SYSTEM DASDA12 (* System Configuration *)
  (* Standard: 61499-1 *)
  (* Version 0.4, 2009-03-05, JHC, Holobloc Inc., Deleted Application. *)
  (* Version 0.3, 2003-12-05, JHC, Rockwell Automation, Renamed from NEWSYSTEM. *)
  (* Version 0.2, 2002-11-05, JHC, Rockwell Automation, Fixed missing (empty) FBD in Application. *)
  (* Version 0.1, 2002-01-17, JHC, Rockwell Automation, Minor cleanup *)
  (* Version 0.0, 2000-05-27, JHC, Rockwell Automation *)
  DEVICE HMI_LAYER : FRAME_DEVICE(BOUNDS := [0,0,200,400])
    RESOURCE HMI : PANEL_RESOURCE(ROWS := 5, COLS := 1)
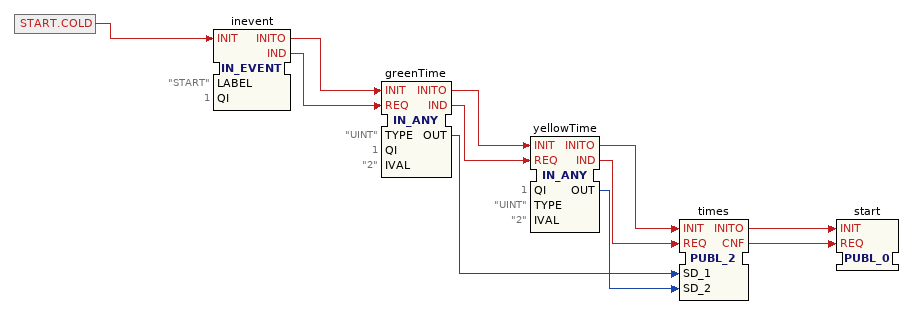
      FBS
        inevent : IN_EVENT(LABEL := "START", QI := 1);
        start : PUBL_0;
        greenTime : IN_ANY(TYPE := "UINT", QI := 1, IVAL := "2");
        yellowTime : IN_ANY(QI := 1, TYPE := "UINT", IVAL := "2");
        times : PUBL_2;
      END_FBS
      EVENT_CONNECTIONS
        START.COLD TO inevent.INIT;
        greenTime.INITO TO yellowTime.INIT;
        inevent.INITO TO greenTime.INIT;
        inevent.IND TO greenTime.REQ;
        yellowTime.INITO TO times.INIT;
        times.INITO TO start.INIT;
        times.CNF TO start.REQ;
        greenTime.IND TO yellowTime.REQ;
        yellowTime.IND TO times.REQ;
      END_CONNECTIONS
      DATA_CONNECTIONS
        greenTime.OUT TO times.SD_1;
        yellowTime.OUT TO times.SD_2;
      END_CONNECTIONS
    END_RESOURCE
  END_DEVICE
  DEVICE MODEL_LAYER : FRAME_DEVICE
    RESOURCE LIGHTS : PANEL_RESOURCE
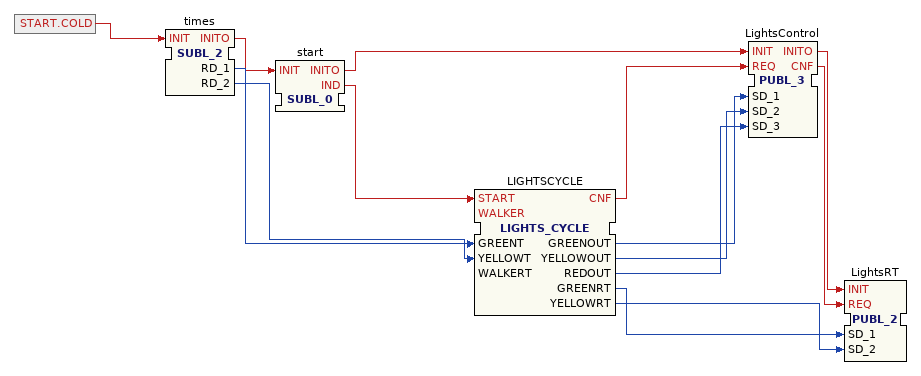
      FBS
        LightsControl : PUBL_3;
        start : SUBL_0;
        times : SUBL_2;
        LIGHTSCYCLE : LIGHTS_CYCLE;
        LightsRT : PUBL_2;
      END_FBS
      EVENT_CONNECTIONS
        START.COLD TO times.INIT;
        times.INITO TO start.INIT;
        start.INITO TO LightsControl.INIT;
        start.IND TO LIGHTSCYCLE.START;
        LIGHTSCYCLE.CNF TO LightsControl.REQ;
        LightsControl.INITO TO LightsRT.INIT;
        LightsControl.CNF TO LightsRT.REQ;
      END_CONNECTIONS
      DATA_CONNECTIONS
        LIGHTSCYCLE.GREENOUT TO LightsControl.SD_1;
        LIGHTSCYCLE.YELLOWOUT TO LightsControl.SD_2;
        LIGHTSCYCLE.REDOUT TO LightsControl.SD_3;
        LIGHTSCYCLE.GREENRT TO LightsRT.SD_1;
        LIGHTSCYCLE.YELLOWRT TO LightsRT.SD_2;
        times.RD_1 TO LIGHTSCYCLE.GREENT;
        times.RD_2 TO LIGHTSCYCLE.YELLOWT;
      END_CONNECTIONS
    END_RESOURCE
  END_DEVICE
  DEVICE VIEW_LAYER : FRAME_DEVICE(BOUNDS := [200,0,600,400], GRID := [1,1])
    RESOURCE view_res : PANEL_RESOURCE
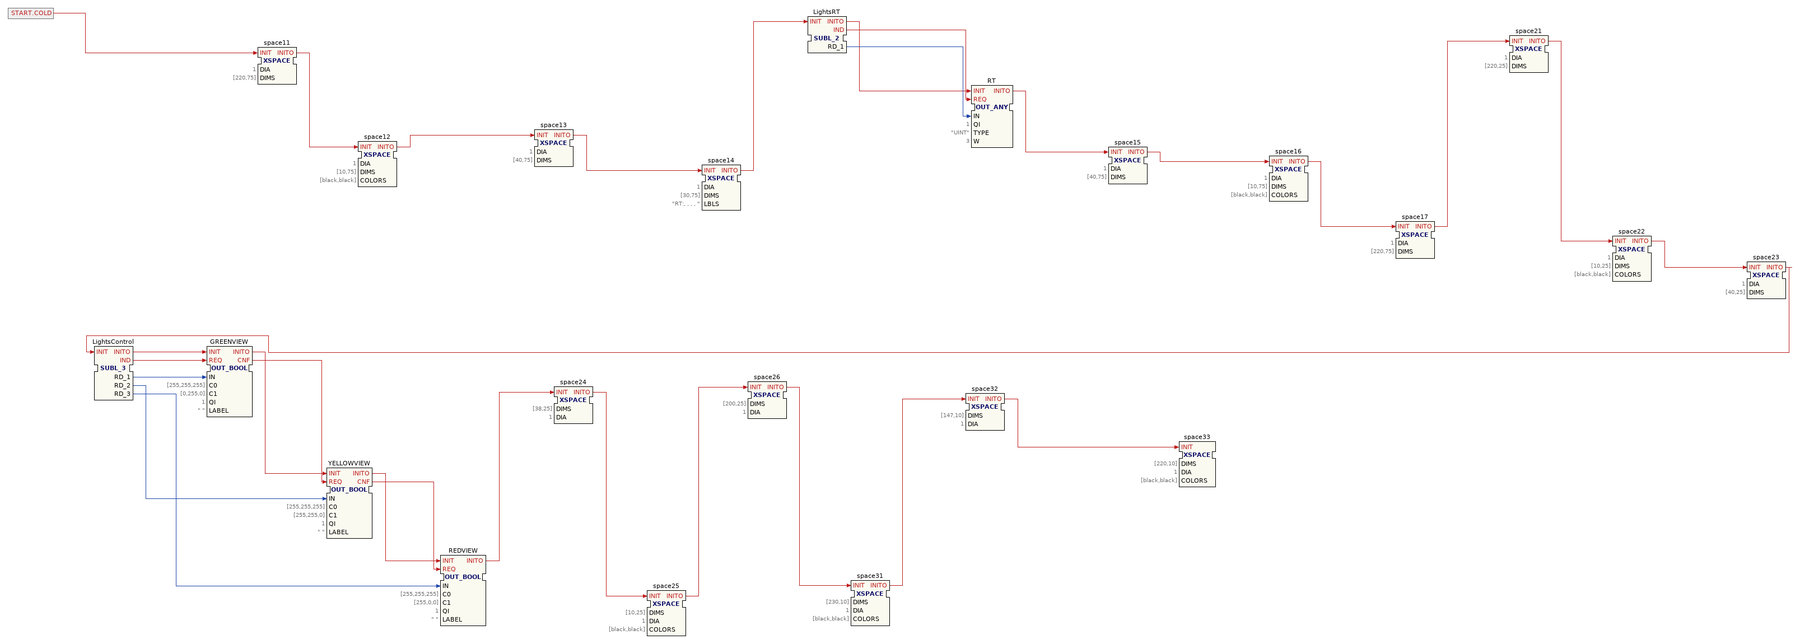
      FBS
        LightsControl : SUBL_3;
        GREENVIEW : OUT_BOOL(C0 := [255,255,255], C1 := [0,255,0], QI := 1, LABEL := " ");
        YELLOWVIEW : OUT_BOOL(C0 := [255,255,255], C1 := [255,255,0], QI := 1, LABEL := " ");
        REDVIEW : OUT_BOOL(C0 := [255,255,255], C1 := [255,0,0], QI := 1, LABEL := " ");
        space11 : XSPACE(DIA := 1, DIMS := [220,75]);
        space12 : XSPACE(DIA := 1, DIMS := [10,75], COLORS := [black,black]);
        space13 : XSPACE(DIA := 1, DIMS := [40,75]);
        space16 : XSPACE(DIA := 1, DIMS := [10,75], COLORS := [black,black]);
        space17 : XSPACE(DIA := 1, DIMS := [220,75]);
        space21 : XSPACE(DIA := 1, DIMS := [220,25]);
        space22 : XSPACE(DIA := 1, DIMS := [10,25], COLORS := [black,black]);
        space23 : XSPACE(DIA := 1, DIMS := [40,25]);
        space24 : XSPACE(DIMS := [38,25], DIA := 1);
        space25 : XSPACE(DIMS := [10,25], DIA := 1, COLORS := [black,black]);
        LightsRT : SUBL_2;
        space14 : XSPACE(DIA := 1, DIMS := [30,75], LBLS := "RT:, , , , ");
        RT : OUT_ANY(QI := 1, TYPE := "UINT", W := 3);
        space15 : XSPACE(DIA := 1, DIMS := [40,75]);
        space26 : XSPACE(DIMS := [200,25], DIA := 1);
        space31 : XSPACE(DIMS := [230,10], DIA := 1, COLORS := [black,black]);
        space32 : XSPACE(DIMS := [147,10], DIA := 1);
        space33 : XSPACE(DIMS := [220,10], DIA := 1, COLORS := [black,black]);
      END_FBS
      EVENT_CONNECTIONS
        LightsControl.INITO TO GREENVIEW.INIT;
        GREENVIEW.INITO TO YELLOWVIEW.INIT;
        YELLOWVIEW.INITO TO REDVIEW.INIT;
        LightsControl.IND TO GREENVIEW.REQ;
        GREENVIEW.CNF TO YELLOWVIEW.REQ;
        YELLOWVIEW.CNF TO REDVIEW.REQ;
        START.COLD TO space11.INIT;
        space11.INITO TO space12.INIT;
        space12.INITO TO space13.INIT;
        space16.INITO TO space17.INIT;
        space17.INITO TO space21.INIT;
        space21.INITO TO space22.INIT;
        space22.INITO TO space23.INIT;
        space23.INITO TO LightsControl.INIT;
        REDVIEW.INITO TO space24.INIT;
        space24.INITO TO space25.INIT;
        space13.INITO TO space14.INIT;
        space14.INITO TO LightsRT.INIT;
        LightsRT.INITO TO RT.INIT;
        LightsRT.IND TO RT.REQ;
        RT.INITO TO space15.INIT;
        space15.INITO TO space16.INIT;
        space25.INITO TO space26.INIT;
        space26.INITO TO space31.INIT;
        space31.INITO TO space32.INIT;
        space32.INITO TO space33.INIT;
      END_CONNECTIONS
      DATA_CONNECTIONS
        LightsControl.RD_1 TO GREENVIEW.IN;
        LightsControl.RD_2 TO YELLOWVIEW.IN;
        LightsControl.RD_3 TO REDVIEW.IN;
        LightsRT.RD_1 TO RT.IN;
      END_CONNECTIONS
    END_RESOURCE
  END_DEVICE
END_SYSTEM
